PROGRAM BH0JPL_LineBackground
VAR
END_VAR

MAIN.stLine_BH0JPL.fbLine(stLine:=MAIN.stLine_BH0JPL);
MAIN.stLine_BH0JPL.stStation_BH0JPL01.fbStation(
				stLine:=MAIN.stLine_BH0JPL,
				stStation:=MAIN.stLine_BH0JPL.stStation_BH0JPL01);

END_PROGRAM

(* stored: Version 1.1.0.1, ProductVersion 3.1.4024.15
   POU BH0JPL_LineBackground: Id {bd9bc2af-56f6-462f-af44-0aefbb87c619}, SpecialFunc None *)
